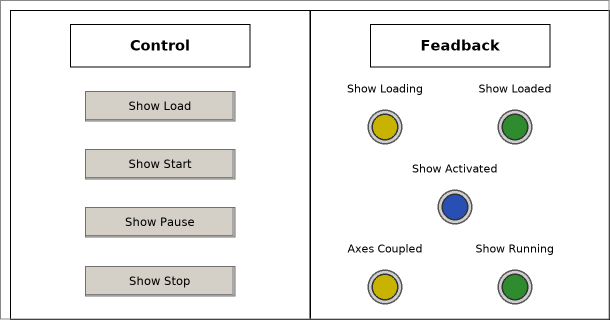
VISUALIZATION Visualization  // 610x320
    Rectangle (310,10 300x310)
    Rectangle (10,10 300x310)
    Button (85,91 150x30), "Show Load", input disabled if: MAIN.boShowActived OR MAIN.fbCsvRead.OUT_boBusy
        tap MAIN.boShowLoad
    Rectangle (70,24 180x43), "Control"
    Button (85,149 150x30), "Show Start", input disabled if: (MAIN.boShowActived AND NOT MAIN.boShowPauseLatch) OR MAIN.fbCsvRead.OUT_boBusy OR NOT MAIN.boShowLoaded
        tap MAIN.boShowStart
    Button (85,207 150x30), "Show Pause", input disabled if: NOT MAIN.fbMasterMoveAbs.Busy
        tap MAIN.boShowPause
    Button (85,266 150x30), "Show Stop", input disabled if: NOT MAIN.fbMasterMoveAbs.Busy
        tap MAIN.boShowStop
    Rectangle (370,24 180x43), "Feadback"
    Lamp1 (365,107 40x40), variable: MAIN.boShowLoading, style: Lamp-Lamp1-Yellow
    Rectangle (335,79 100x20), "Show Loading"
    Lamp1 (495,107 40x40), variable: MAIN.boShowLoaded, style: Lamp-Lamp1-Green
    Rectangle (465,79 100x20), "Show Loaded"
    Lamp1 (435,187 40x40), variable: MAIN.boShowActived, style: Lamp-Lamp1-Blue
    Rectangle (405,159 100x20), "Show Activated"
    Lamp1 (365,267 40x40), variable: MAIN.AXMaster.NcToPlc.CoupleState = 1, style: Lamp-Lamp1-Yellow
    Rectangle (335,239 100x20), "Axes Coupled"
    Lamp1 (495,267 40x40), variable: MAIN.fbMasterMoveAbs.Busy, style: Lamp-Lamp1-Green
    Rectangle (465,239 100x20), "Show Running"
END_VISUALIZATION

(* stored: Version 1.1.0.1, ProductVersion 3.1.4024.12
   Visu Visualization: Id {5104f3be-746c-4969-baf8-5a1a1439efaf} *)
